// TIA Portal project "Conveyor_Robot_Backup_01_04_2026_V17" (V17)

(* hardware
DEVICE "S7-1200 station_1"  S7-1200 Station
   slot 0: "Rack_0"  S7-1200 Rack  Rack  V1.0
   slot 1: "PLC_1"  CPU 1214C DC/DC/DC  6ES7 214-1AG40-0XB0  V4.4
   slot 2: "DI 8x24VDC/DQ 8xRelay_1"  SM 1223 DI8/DQ8 x relay  6ES7 223-1PH32-0XB0  V2.0
   slot 3: "DI 8x24VDC/DQ 8xRelay_2"  SM 1223 DI8/DQ8 x relay  6ES7 223-1PH32-0XB0  V2.0
DEVICE "HMI_1"  KTP700 Basic PN
   slot 0: "HMI_1"  KTP700 Basic PN  6AV2 123-2GB03-0AX0  16.0.0.0
   slot 1: "HMI_RT_1"  KTP700 Basic PN  6AV2 123-2GB03-0AX0  16.0.0.0
   slot 5: "HMI_1.IE_CP_1"  PROFINET Interface  16.0.0.0
      slot 1: "PROFINET Interface_1"  PROFINET Interface
         slot 1: "Port_1"  Port
*)

// ===== PLC "PLC_1"  CPU 1214C DC/DC/DC =====

VAR_GLOBAL   // PLC tag table "Default tag table"
   "I_PB_Start" AT %I0.0 : Bool;
   "I_PB_Stop" AT %I0.1 : Bool;
   "I_PB_Emergency" AT %I0.2 : Bool;
   "I_PB_Reset" AT %I0.3 : Bool;
   "I_PB_Auto" AT %I0.4 : Bool;
   "I_Sensor_Entry" AT %I0.5 : Bool;
   "I_Sensor_Weigh" AT %I0.6 : Bool;
   "I_Sensor_Decision" AT %I0.7 : Bool;
   "I_Sensor_Reject" AT %I1.0 : Bool;
   "I_Sensor_Exit" AT %I1.1 : Bool;
   "I_Pusher_Extend" AT %I1.2 : Bool;
   "I_Pusher_Released" AT %I1.3 : Bool;
   "I_OL_EntryMotor" AT %I1.4 : Bool;
   "I_OL_WeighMotor" AT %I1.5 : Bool;
   "I_OL_DecideMotor" AT %I2.0 : Bool;
   "I_OL_RejectMotor" AT %I2.1 : Bool;
   "I_OL_ExitMotor" AT %I2.2 : Bool;
   "I_Robot_Detect" AT %I2.3 : Bool;
   "I_Robot_Moving_X" AT %I2.4 : Bool;
   "I_Robot_Moving_Z" AT %I2.5 : Bool;
   "I_Robot_Rotating" AT %I2.6 : Bool;
   "IW_Weight_Loadcell" AT %ID30 : Real;
   "Q_Motor_Entry" AT %Q0.0 : Bool;
   "Q_Motor_Weigh" AT %Q0.1 : Bool;
   "Q_Motor_Decision" AT %Q0.2 : Bool;
   "Q_Motor_reject" AT %Q0.3 : Bool;
   "Q_Motor_Exit" AT %Q0.4 : Bool;
   "Q_Pusher_Extend" AT %Q0.5 : Bool;
   "Q_Pusher_Release" AT %Q0.6 : Bool;
   "Q_Signal_Red" AT %Q2.0 : Bool;
   "Q_Signal_Yellow" AT %Q0.7 : Bool;
   "Q_Signal_Green" AT %Q2.1 : Bool;
   "Q_Buzzer" AT %Q2.2 : Bool;
   "Q_Robot_Extend_X" AT %Q2.3 : Bool;
   "Q_Robot_Down_Z" AT %Q2.4 : Bool;
   "Q_Robot_Grab" AT %Q2.5 : Bool;
   "Q_Robot_Rotate_CW" AT %Q2.6 : Bool;
   "Q_Robot_Rotate_CCW" AT %Q2.7 : Bool;
   "System_Byte" AT %MB1 : Byte;
   "FirstScan" AT %M1.0 : Bool;
   "DiagStatusUpdate" AT %M1.1 : Bool;
   "AlwaysTRUE" AT %M1.2 : Bool;
   "AlwaysFALSE" AT %M1.3 : Bool;
   "Clock_Byte" AT %MB50 : Byte;
   "Clock_10Hz" AT %M50.0 : Bool;
   "Clock_5Hz" AT %M50.1 : Bool;
   "Clock_2.5Hz" AT %M50.2 : Bool;
   "Clock_2Hz" AT %M50.3 : Bool;
   "Clock_1.25Hz" AT %M50.4 : Bool;
   "Clock_1Hz" AT %M50.5 : Bool;
   "Clock_0.625Hz" AT %M50.6 : Bool;
   "Clock_0.5Hz" AT %M50.7 : Bool;
END_VAR

TYPE "UDT_Box_Data"
   STRUCT
      BoxId : Int;
      Weight : Real;
      Status : Bool;
   END_STRUCT;
END_TYPE

TYPE "UDT_Box_Real_Data"
   STRUCT
      Actual_Weight_Value : Real;
      Accept_Limit_Low : Real;
      Accept_Limit_High : Real;
      Current_Box_ID : Int;
   END_STRUCT;
END_TYPE

TYPE "UDT_Alarm"
   STRUCT
      Active : Bool;
      Acknowledge : Bool;
      Cleared : Bool;
      TimeStamp : DTL;
      Duration : Time;
   END_STRUCT;
END_TYPE

TYPE "UDT_OEE_Data"
   STRUCT
      Availability : Real;
      Quality : Real;
      Overall : Real;
      Rating : String;
      Accept_Ratio : Real;
      Reject_Ratio : Real;
   END_STRUCT;
END_TYPE

// folder: 01_Global_DBs

DATA_BLOCK "DB_Batch_Data"   // DB2
{ S7_Optimized_Access := 'TRUE' }
VERSION : 0.1
   VAR
      Batch_ID : Int;
      Batch_Boxes : Int;
      Accept_Boxes : Int;
      Reject_Boxes : Int;
      Accept_Total_Weight : Real;
      Reject_Total_Weight : Real;
      Batch_Running : Bool;
      Low_Limit_Tag : Real;
      High_Limit_Tag : Real;
      Low_Limit_Tag_1 : Real;
      High_Limit_Tag_1 : Real;
      Real_Box_Data : "UDT_Box_Real_Data";
      OEE_Data : "UDT_OEE_Data";
   END_VAR
BEGIN
   Real_Box_Data.Accept_Limit_Low := 3.0;
   Real_Box_Data.Accept_Limit_High := 6.0;
   Real_Box_Data.Current_Box_ID := 0;
END_DATA_BLOCK

DATA_BLOCK "DB_Alarms"   // DB9
{ S7_Optimized_Access := 'TRUE' }
VERSION : 0.1
   VAR
      Motor_Overload : Struct
         OL_EntryMotor : "UDT_Alarm";
         OL_WeighMotor : "UDT_Alarm";
         OL_DecisionMotor : "UDT_Alarm";
         OL_RejectMotor : "UDT_Alarm";
         OL_ExitMotor : "UDT_Alarm";
      END_STRUCT;
      Jam_Alarm : Struct
         Jam_EntryMotor : "UDT_Alarm";
         Jam_WeighMotor : "UDT_Alarm";
         Jam_DecisionMotor : "UDT_Alarm";
         Jam_RejectMotor : "UDT_Alarm";
         Jam_ExitMotor : "UDT_Alarm";
      END_STRUCT;
      Pusher_Alarm : Struct
         Pusher_Stuck_Extended : "UDT_Alarm";
         Pusher_Stuck_Retracted : "UDT_Alarm";
      END_STRUCT;
      HMI_Alarm : Struct
         Jam_Alarm : Word;
         OL_Alarm : Word;
         System_Alarm : Word;
      END_STRUCT;
      HMI_Ack_All : Bool;
   END_VAR
BEGIN
END_DATA_BLOCK

DATA_BLOCK "DB_System_Status"   // DB12
{ S7_Optimized_Access := 'TRUE' }
VERSION : 0.1
   VAR
      System_Running : Bool;
      Enable_Entry : Bool;
      Enable_Weigh : Bool;
      Enable_Decision : Bool;
      Enable_Reject : Bool;
      Enable_Exit : Bool;
      Enable_Robot : Bool;
      Jam_Detected : Struct
         Entry_Jam_Detected : Bool;
         Weigh_Jam_Detected : Bool;
         Decision_Jam_Detected : Bool;
         Reject_Jam_Detected : Bool;
         Exit_Jam_Detected : Bool;
      END_STRUCT;
   END_VAR
BEGIN
END_DATA_BLOCK

// folder: 04_Application_Blocks

DATA_BLOCK "Motor_Control_DB_Entry"   // DB3
{ S7_Optimized_Access := 'TRUE' }
VERSION : 0.1
// stored: InstanceOfName Motor_Control
"Motor_Control"
BEGIN
END_DATA_BLOCK

DATA_BLOCK "Motor_Control_DB_Weigh"   // DB4
{ S7_Optimized_Access := 'TRUE' }
VERSION : 0.1
// stored: InstanceOfName Motor_Control
"Motor_Control"
BEGIN
END_DATA_BLOCK

DATA_BLOCK "Motor_Control_DB_Decision"   // DB5
{ S7_Optimized_Access := 'TRUE' }
VERSION : 0.1
// stored: InstanceOfName Motor_Control
"Motor_Control"
BEGIN
END_DATA_BLOCK

DATA_BLOCK "Motor_Control_DB_Exit"   // DB6
{ S7_Optimized_Access := 'TRUE' }
VERSION : 0.1
// stored: InstanceOfName Motor_Control
"Motor_Control"
BEGIN
END_DATA_BLOCK

DATA_BLOCK "Reject_Conveyor_Control_DB"   // DB7
{ S7_Optimized_Access := 'TRUE' }
VERSION : 0.1
// stored: InstanceOfName Reject_Conveyor_Control
"Reject_Conveyor_Control"
BEGIN
END_DATA_BLOCK

DATA_BLOCK "Arm_Pick_&_Place_DB"   // DB8
{ S7_Optimized_Access := 'TRUE' }
VERSION : 0.1
// stored: InstanceOfName Arm_Pick_&_Place
"Arm_Pick_&_Place"
BEGIN
END_DATA_BLOCK

// folder: 06_IO_Mapping

DATA_BLOCK "DB_IO_Mapping"   // DB1
{ S7_Optimized_Access := 'TRUE' }
VERSION : 0.1
   VAR
      Input : Struct
         I_PB_Start : Bool;
         I_PB_Stop : Bool;
         I_PB_Emergency : Bool;
         I_PB_Reset : Bool;
         I_PB_Auto : Bool;
         I_Sensor_Entry : Bool;
         I_Sensor_Weigh : Bool;
         I_Sensor_Decision : Bool;
         I_Sensor_Reject : Bool;
         I_Sensor_Exit : Bool;
         I_Pusher_Extend : Bool;
         I_Pusher_Released : Bool;
         I_OL_EntryMotor : Bool;
         I_OL_WeighMotor : Bool;
         I_OL_DecideMotor : Bool;
         I_OL_RejectMotor : Bool;
         I_OL_ExitMotor : Bool;
         I_Robot_Detect : Bool;
         I_Robot_Moving_X : Bool;
         I_Robot_Moving_Z : Bool;
         I_Robot_Rotating : Bool;
         IW_Weight_Loadcell : Real;
      END_STRUCT;
      Output : Struct
         Q_Motor_Entry : Bool;
         Q_Motor_Weigh : Bool;
         Q_Motor_Decision : Bool;
         Q_Motor_reject : Bool;
         Q_Motor_Exit : Bool;
         Q_Pusher_Extend : Bool;
         Q_Pusher_Release : Bool;
         Q_Signal_Red : Bool;
         Q_Signal_Yellow : Bool;
         Q_Signal_Green : Bool;
         Q_Buzzer : Bool;
         Q_Robot_Extend_X : Bool;
         Q_Robot_Down_Z : Bool;
         Q_Robot_Grab : Bool;
         Q_Robot_Rotate_CW : Bool;
         Q_Robot_Rotate_CCW : Bool;
      END_STRUCT;
      Parameter : Struct
         M_START : Bool;
      END_STRUCT;
   END_VAR
BEGIN
END_DATA_BLOCK

// folder: System blocks/Program resources

DATA_BLOCK "IEC_Timer_0_DB_1"   // DB10
{ S7_Optimized_Access := 'TRUE' }
AUTHOR : Simatic
FAMILY : IEC
NAME : IEC_TMR
VERSION : 1.0
// stored: InstanceOfName IEC_TIMER
"IEC_TIMER"
BEGIN
END_DATA_BLOCK

// folder: 00_System_Blocks

ORGANIZATION_BLOCK "Main"   // OB1, LAD, ProgramCycle
TITLE = "Main Program Sweep (Cycle)"
{ S7_Optimized_Access := 'TRUE' }
VERSION : 0.1
   VAR_INPUT
      Initial_Call : Bool;   // Initial call of this OB
      Remanence : Bool;   // =True, if remanent data are available
   END_VAR
BEGIN

REGION Network 1: Factory IO Interface
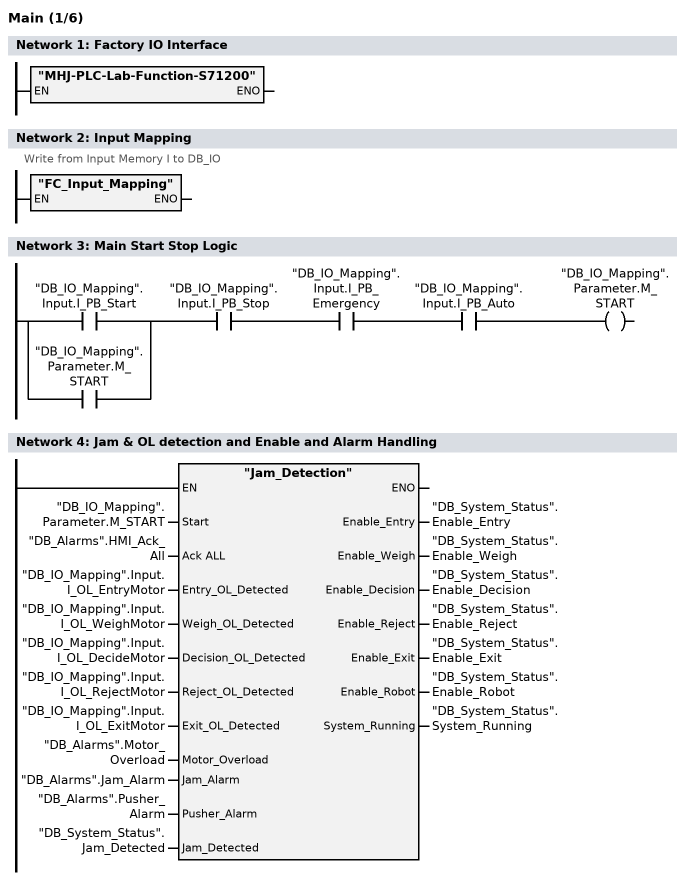
   RUNG wire#powerrail
      "MHJ-PLC-Lab-Function-S71200"()
   END_RUNG
   // the same network as SCL:
   "MHJ-PLC-Lab-Function-S71200"();
END_REGION

REGION Network 2: Input Mapping
   // Write from Input Memory I to DB_IO
   RUNG wire#powerrail
      "FC_Input_Mapping"()
   END_RUNG
   // the same network as SCL:
   "FC_Input_Mapping"();
END_REGION

REGION Network 3: Main Start Stop Logic
   RUNG wire#powerrail
      Contact( "DB_IO_Mapping".Input.I_PB_Start )
      wire#w1
      Contact( "DB_IO_Mapping".Input.I_PB_Stop )
      Contact( "DB_IO_Mapping".Input.I_PB_Emergency )
      Contact( "DB_IO_Mapping".Input.I_PB_Auto )
      Coil( "DB_IO_Mapping".Parameter.M_START )
   END_RUNG
   RUNG wire#powerrail
      Contact( "DB_IO_Mapping".Parameter.M_START )
   END_RUNG wire#w1
   // the same network as SCL:
   "DB_IO_Mapping".Parameter.M_START := ("DB_IO_Mapping".Input.I_PB_Start OR "DB_IO_Mapping".Parameter.M_START) AND "DB_IO_Mapping".Input.I_PB_Stop AND "DB_IO_Mapping".Input.I_PB_Emergency AND "DB_IO_Mapping".Input.I_PB_Auto;
END_REGION

REGION Network 4: Jam & OL detection and Enable and Alarm Handling
   RUNG wire#powerrail
      "Jam_Detection"(Start := "DB_IO_Mapping".Parameter.M_START, "Ack ALL" := "DB_Alarms".HMI_Ack_All, Entry_OL_Detected := "DB_IO_Mapping".Input.I_OL_EntryMotor, Weigh_OL_Detected := "DB_IO_Mapping".Input.I_OL_WeighMotor, Decision_OL_Detected := "DB_IO_Mapping".Input.I_OL_DecideMotor, Reject_OL_Detected := "DB_IO_Mapping".Input.I_OL_RejectMotor, Exit_OL_Detected := "DB_IO_Mapping".Input.I_OL_ExitMotor, Motor_Overload := "DB_Alarms".Motor_Overload, Jam_Alarm := "DB_Alarms".Jam_Alarm, Pusher_Alarm := "DB_Alarms".Pusher_Alarm, Jam_Detected := "DB_System_Status".Jam_Detected, Enable_Entry => "DB_System_Status".Enable_Entry, Enable_Weigh => "DB_System_Status".Enable_Weigh, Enable_Decision => "DB_System_Status".Enable_Decision, Enable_Reject => "DB_System_Status".Enable_Reject, Enable_Exit => "DB_System_Status".Enable_Exit, Enable_Robot => "DB_System_Status".Enable_Robot, System_Running => "DB_System_Status".System_Running)
   END_RUNG
   // the same network as SCL:
   "Jam_Detection"(Start := "DB_IO_Mapping".Parameter.M_START,
                   "Ack ALL" := "DB_Alarms".HMI_Ack_All,
                   Entry_OL_Detected := "DB_IO_Mapping".Input.I_OL_EntryMotor,
                   Weigh_OL_Detected := "DB_IO_Mapping".Input.I_OL_WeighMotor,
                   Decision_OL_Detected := "DB_IO_Mapping".Input.I_OL_DecideMotor,
                   Reject_OL_Detected := "DB_IO_Mapping".Input.I_OL_RejectMotor,
                   Exit_OL_Detected := "DB_IO_Mapping".Input.I_OL_ExitMotor,
                   Motor_Overload := "DB_Alarms".Motor_Overload,
                   Jam_Alarm := "DB_Alarms".Jam_Alarm,
                   Pusher_Alarm := "DB_Alarms".Pusher_Alarm,
                   Jam_Detected := "DB_System_Status".Jam_Detected,
                   Enable_Entry => "DB_System_Status".Enable_Entry,
                   Enable_Weigh => "DB_System_Status".Enable_Weigh,
                   Enable_Decision => "DB_System_Status".Enable_Decision,
                   Enable_Reject => "DB_System_Status".Enable_Reject,
                   Enable_Exit => "DB_System_Status".Enable_Exit,
                   Enable_Robot => "DB_System_Status".Enable_Robot,
                   System_Running => "DB_System_Status".System_Running);
END_REGION

REGION Network 5: Entry Conveyor
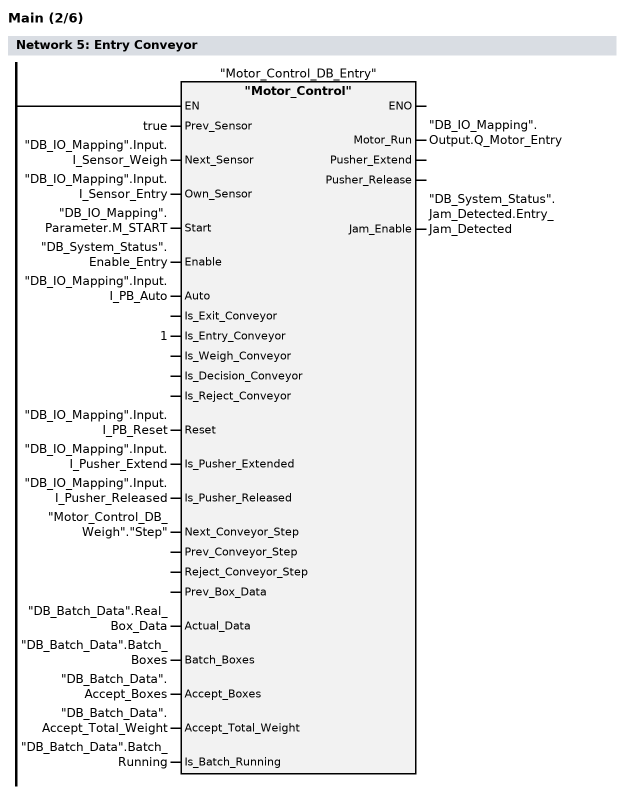
   RUNG wire#powerrail
      "Motor_Control_DB_Entry"(Prev_Sensor := true, Next_Sensor := "DB_IO_Mapping".Input.I_Sensor_Weigh, Own_Sensor := "DB_IO_Mapping".Input.I_Sensor_Entry, Start := "DB_IO_Mapping".Parameter.M_START, Enable := "DB_System_Status".Enable_Entry, Auto := "DB_IO_Mapping".Input.I_PB_Auto, Is_Exit_Conveyor :=, Is_Entry_Conveyor := 1, Is_Weigh_Conveyor :=, Is_Decision_Conveyor :=, Is_Reject_Conveyor :=, Reset := "DB_IO_Mapping".Input.I_PB_Reset, Is_Pusher_Extended := "DB_IO_Mapping".Input.I_Pusher_Extend, Is_Pusher_Released := "DB_IO_Mapping".Input.I_Pusher_Released, Next_Conveyor_Step := "Motor_Control_DB_Weigh"."Step", Prev_Conveyor_Step :=, Reject_Conveyor_Step :=, Prev_Box_Data :=, Actual_Data := "DB_Batch_Data".Real_Box_Data, Batch_Boxes := "DB_Batch_Data".Batch_Boxes, Accept_Boxes := "DB_Batch_Data".Accept_Boxes, Accept_Total_Weight := "DB_Batch_Data".Accept_Total_Weight, Is_Batch_Running := "DB_Batch_Data".Batch_Running, Motor_Run => "DB_IO_Mapping".Output.Q_Motor_Entry, Pusher_Extend =>, Pusher_Release =>, Jam_Enable => "DB_System_Status".Jam_Detected.Entry_Jam_Detected)
   END_RUNG
   // the same network as SCL:
   "Motor_Control_DB_Entry"(Prev_Sensor := true,   // "Motor_Control"
                           Next_Sensor := "DB_IO_Mapping".Input.I_Sensor_Weigh,
                           Own_Sensor := "DB_IO_Mapping".Input.I_Sensor_Entry,
                           Start := "DB_IO_Mapping".Parameter.M_START,
                           Enable := "DB_System_Status".Enable_Entry,
                           Auto := "DB_IO_Mapping".Input.I_PB_Auto,
                           Is_Entry_Conveyor := 1,
                           Reset := "DB_IO_Mapping".Input.I_PB_Reset,
                           Is_Pusher_Extended := "DB_IO_Mapping".Input.I_Pusher_Extend,
                           Is_Pusher_Released := "DB_IO_Mapping".Input.I_Pusher_Released,
                           Next_Conveyor_Step := "Motor_Control_DB_Weigh"."Step",
                           Actual_Data := "DB_Batch_Data".Real_Box_Data,
                           Batch_Boxes := "DB_Batch_Data".Batch_Boxes,
                           Accept_Boxes := "DB_Batch_Data".Accept_Boxes,
                           Accept_Total_Weight := "DB_Batch_Data".Accept_Total_Weight,
                           Is_Batch_Running := "DB_Batch_Data".Batch_Running,
                           Motor_Run => "DB_IO_Mapping".Output.Q_Motor_Entry,
                           Jam_Enable => "DB_System_Status".Jam_Detected.Entry_Jam_Detected);
END_REGION

REGION Network 6: Weigh Conveyor
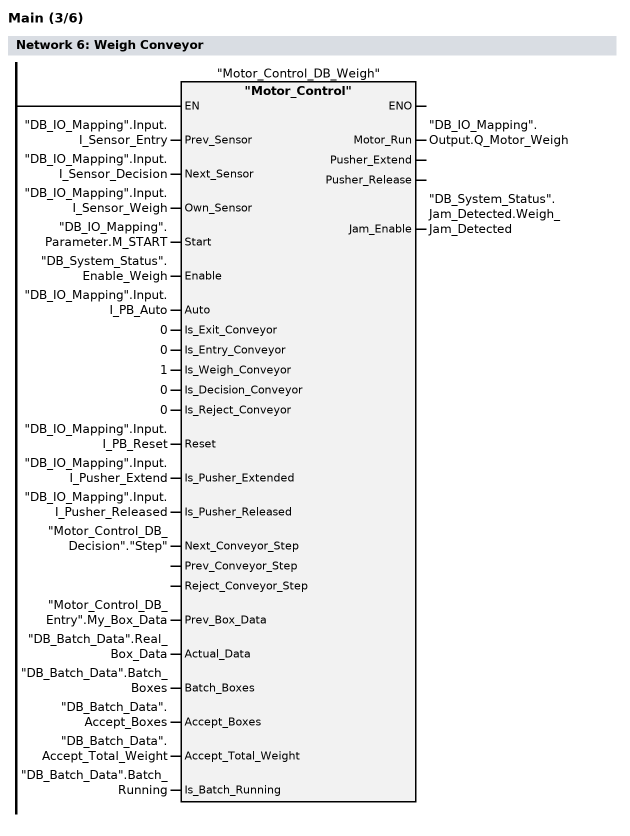
   RUNG wire#powerrail
      "Motor_Control_DB_Weigh"(Prev_Sensor := "DB_IO_Mapping".Input.I_Sensor_Entry, Next_Sensor := "DB_IO_Mapping".Input.I_Sensor_Decision, Own_Sensor := "DB_IO_Mapping".Input.I_Sensor_Weigh, Start := "DB_IO_Mapping".Parameter.M_START, Enable := "DB_System_Status".Enable_Weigh, Auto := "DB_IO_Mapping".Input.I_PB_Auto, Is_Exit_Conveyor := 0, Is_Entry_Conveyor := 0, Is_Weigh_Conveyor := 1, Is_Decision_Conveyor := 0, Is_Reject_Conveyor := 0, Reset := "DB_IO_Mapping".Input.I_PB_Reset, Is_Pusher_Extended := "DB_IO_Mapping".Input.I_Pusher_Extend, Is_Pusher_Released := "DB_IO_Mapping".Input.I_Pusher_Released, Next_Conveyor_Step := "Motor_Control_DB_Decision"."Step", Prev_Conveyor_Step :=, Reject_Conveyor_Step :=, Prev_Box_Data := "Motor_Control_DB_Entry".My_Box_Data, Actual_Data := "DB_Batch_Data".Real_Box_Data, Batch_Boxes := "DB_Batch_Data".Batch_Boxes, Accept_Boxes := "DB_Batch_Data".Accept_Boxes, Accept_Total_Weight := "DB_Batch_Data".Accept_Total_Weight, Is_Batch_Running := "DB_Batch_Data".Batch_Running, Motor_Run => "DB_IO_Mapping".Output.Q_Motor_Weigh, Pusher_Extend =>, Pusher_Release =>, Jam_Enable => "DB_System_Status".Jam_Detected.Weigh_Jam_Detected)
   END_RUNG
   // the same network as SCL:
   "Motor_Control_DB_Weigh"(Prev_Sensor := "DB_IO_Mapping".Input.I_Sensor_Entry,   // "Motor_Control"
                           Next_Sensor := "DB_IO_Mapping".Input.I_Sensor_Decision,
                           Own_Sensor := "DB_IO_Mapping".Input.I_Sensor_Weigh,
                           Start := "DB_IO_Mapping".Parameter.M_START,
                           Enable := "DB_System_Status".Enable_Weigh,
                           Auto := "DB_IO_Mapping".Input.I_PB_Auto,
                           Is_Exit_Conveyor := 0,
                           Is_Entry_Conveyor := 0,
                           Is_Weigh_Conveyor := 1,
                           Is_Decision_Conveyor := 0,
                           Is_Reject_Conveyor := 0,
                           Reset := "DB_IO_Mapping".Input.I_PB_Reset,
                           Is_Pusher_Extended := "DB_IO_Mapping".Input.I_Pusher_Extend,
                           Is_Pusher_Released := "DB_IO_Mapping".Input.I_Pusher_Released,
                           Next_Conveyor_Step := "Motor_Control_DB_Decision"."Step",
                           Prev_Box_Data := "Motor_Control_DB_Entry".My_Box_Data,
                           Actual_Data := "DB_Batch_Data".Real_Box_Data,
                           Batch_Boxes := "DB_Batch_Data".Batch_Boxes,
                           Accept_Boxes := "DB_Batch_Data".Accept_Boxes,
                           Accept_Total_Weight := "DB_Batch_Data".Accept_Total_Weight,
                           Is_Batch_Running := "DB_Batch_Data".Batch_Running,
                           Motor_Run => "DB_IO_Mapping".Output.Q_Motor_Weigh,
                           Jam_Enable => "DB_System_Status".Jam_Detected.Weigh_Jam_Detected);
END_REGION

REGION Network 7: Decision Conveyor
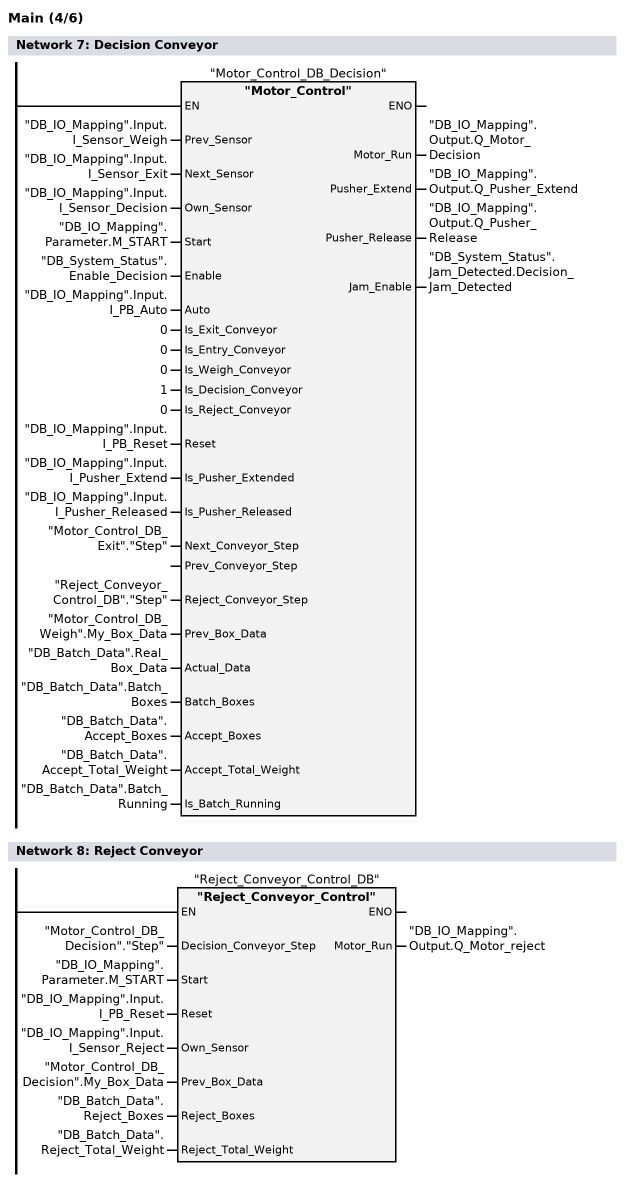
   RUNG wire#powerrail
      "Motor_Control_DB_Decision"(Prev_Sensor := "DB_IO_Mapping".Input.I_Sensor_Weigh, Next_Sensor := "DB_IO_Mapping".Input.I_Sensor_Exit, Own_Sensor := "DB_IO_Mapping".Input.I_Sensor_Decision, Start := "DB_IO_Mapping".Parameter.M_START, Enable := "DB_System_Status".Enable_Decision, Auto := "DB_IO_Mapping".Input.I_PB_Auto, Is_Exit_Conveyor := 0, Is_Entry_Conveyor := 0, Is_Weigh_Conveyor := 0, Is_Decision_Conveyor := 1, Is_Reject_Conveyor := 0, Reset := "DB_IO_Mapping".Input.I_PB_Reset, Is_Pusher_Extended := "DB_IO_Mapping".Input.I_Pusher_Extend, Is_Pusher_Released := "DB_IO_Mapping".Input.I_Pusher_Released, Next_Conveyor_Step := "Motor_Control_DB_Exit"."Step", Prev_Conveyor_Step :=, Reject_Conveyor_Step := "Reject_Conveyor_Control_DB"."Step", Prev_Box_Data := "Motor_Control_DB_Weigh".My_Box_Data, Actual_Data := "DB_Batch_Data".Real_Box_Data, Batch_Boxes := "DB_Batch_Data".Batch_Boxes, Accept_Boxes := "DB_Batch_Data".Accept_Boxes, Accept_Total_Weight := "DB_Batch_Data".Accept_Total_Weight, Is_Batch_Running := "DB_Batch_Data".Batch_Running, Motor_Run => "DB_IO_Mapping".Output.Q_Motor_Decision, Pusher_Extend => "DB_IO_Mapping".Output.Q_Pusher_Extend, Pusher_Release => "DB_IO_Mapping".Output.Q_Pusher_Release, Jam_Enable => "DB_System_Status".Jam_Detected.Decision_Jam_Detected)
   END_RUNG
   // the same network as SCL:
   "Motor_Control_DB_Decision"(Prev_Sensor := "DB_IO_Mapping".Input.I_Sensor_Weigh,   // "Motor_Control"
                           Next_Sensor := "DB_IO_Mapping".Input.I_Sensor_Exit,
                           Own_Sensor := "DB_IO_Mapping".Input.I_Sensor_Decision,
                           Start := "DB_IO_Mapping".Parameter.M_START,
                           Enable := "DB_System_Status".Enable_Decision,
                           Auto := "DB_IO_Mapping".Input.I_PB_Auto,
                           Is_Exit_Conveyor := 0,
                           Is_Entry_Conveyor := 0,
                           Is_Weigh_Conveyor := 0,
                           Is_Decision_Conveyor := 1,
                           Is_Reject_Conveyor := 0,
                           Reset := "DB_IO_Mapping".Input.I_PB_Reset,
                           Is_Pusher_Extended := "DB_IO_Mapping".Input.I_Pusher_Extend,
                           Is_Pusher_Released := "DB_IO_Mapping".Input.I_Pusher_Released,
                           Next_Conveyor_Step := "Motor_Control_DB_Exit"."Step",
                           Reject_Conveyor_Step := "Reject_Conveyor_Control_DB"."Step",
                           Prev_Box_Data := "Motor_Control_DB_Weigh".My_Box_Data,
                           Actual_Data := "DB_Batch_Data".Real_Box_Data,
                           Batch_Boxes := "DB_Batch_Data".Batch_Boxes,
                           Accept_Boxes := "DB_Batch_Data".Accept_Boxes,
                           Accept_Total_Weight := "DB_Batch_Data".Accept_Total_Weight,
                           Is_Batch_Running := "DB_Batch_Data".Batch_Running,
                           Motor_Run => "DB_IO_Mapping".Output.Q_Motor_Decision,
                           Pusher_Extend => "DB_IO_Mapping".Output.Q_Pusher_Extend,
                           Pusher_Release => "DB_IO_Mapping".Output.Q_Pusher_Release,
                           Jam_Enable => "DB_System_Status".Jam_Detected.Decision_Jam_Detected);
END_REGION

REGION Network 8: Reject Conveyor
   RUNG wire#powerrail
      "Reject_Conveyor_Control_DB"(Decision_Conveyor_Step := "Motor_Control_DB_Decision"."Step", Start := "DB_IO_Mapping".Parameter.M_START, Reset := "DB_IO_Mapping".Input.I_PB_Reset, Own_Sensor := "DB_IO_Mapping".Input.I_Sensor_Reject, Prev_Box_Data := "Motor_Control_DB_Decision".My_Box_Data, Reject_Boxes := "DB_Batch_Data".Reject_Boxes, Reject_Total_Weight := "DB_Batch_Data".Reject_Total_Weight, Motor_Run => "DB_IO_Mapping".Output.Q_Motor_reject)
   END_RUNG
   // the same network as SCL:
   "Reject_Conveyor_Control_DB"(Decision_Conveyor_Step := "Motor_Control_DB_Decision"."Step",   // "Reject_Conveyor_Control"
                           Start := "DB_IO_Mapping".Parameter.M_START,
                           Reset := "DB_IO_Mapping".Input.I_PB_Reset,
                           Own_Sensor := "DB_IO_Mapping".Input.I_Sensor_Reject,
                           Prev_Box_Data := "Motor_Control_DB_Decision".My_Box_Data,
                           Reject_Boxes := "DB_Batch_Data".Reject_Boxes,
                           Reject_Total_Weight := "DB_Batch_Data".Reject_Total_Weight,
                           Motor_Run => "DB_IO_Mapping".Output.Q_Motor_reject);
END_REGION

REGION Network 9: Exit Conveyor
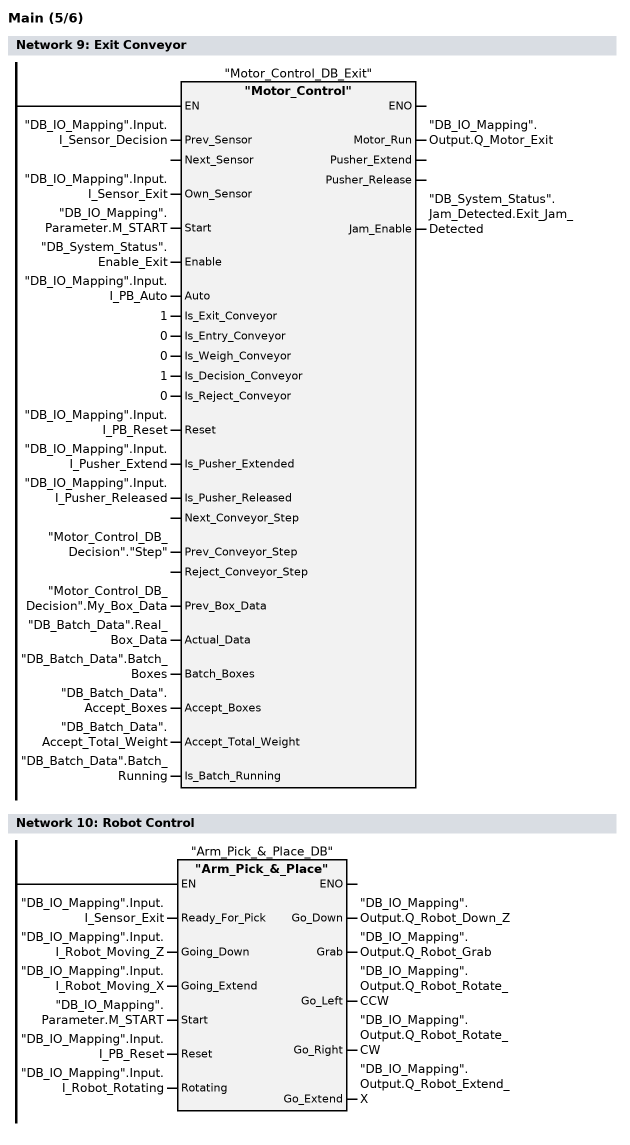
   RUNG wire#powerrail
      "Motor_Control_DB_Exit"(Prev_Sensor := "DB_IO_Mapping".Input.I_Sensor_Decision, Next_Sensor :=, Own_Sensor := "DB_IO_Mapping".Input.I_Sensor_Exit, Start := "DB_IO_Mapping".Parameter.M_START, Enable := "DB_System_Status".Enable_Exit, Auto := "DB_IO_Mapping".Input.I_PB_Auto, Is_Exit_Conveyor := 1, Is_Entry_Conveyor := 0, Is_Weigh_Conveyor := 0, Is_Decision_Conveyor := 1, Is_Reject_Conveyor := 0, Reset := "DB_IO_Mapping".Input.I_PB_Reset, Is_Pusher_Extended := "DB_IO_Mapping".Input.I_Pusher_Extend, Is_Pusher_Released := "DB_IO_Mapping".Input.I_Pusher_Released, Next_Conveyor_Step :=, Prev_Conveyor_Step := "Motor_Control_DB_Decision"."Step", Reject_Conveyor_Step :=, Prev_Box_Data := "Motor_Control_DB_Decision".My_Box_Data, Actual_Data := "DB_Batch_Data".Real_Box_Data, Batch_Boxes := "DB_Batch_Data".Batch_Boxes, Accept_Boxes := "DB_Batch_Data".Accept_Boxes, Accept_Total_Weight := "DB_Batch_Data".Accept_Total_Weight, Is_Batch_Running := "DB_Batch_Data".Batch_Running, Motor_Run => "DB_IO_Mapping".Output.Q_Motor_Exit, Pusher_Extend =>, Pusher_Release =>, Jam_Enable => "DB_System_Status".Jam_Detected.Exit_Jam_Detected)
   END_RUNG
   // the same network as SCL:
   "Motor_Control_DB_Exit"(Prev_Sensor := "DB_IO_Mapping".Input.I_Sensor_Decision,   // "Motor_Control"
                           Own_Sensor := "DB_IO_Mapping".Input.I_Sensor_Exit,
                           Start := "DB_IO_Mapping".Parameter.M_START,
                           Enable := "DB_System_Status".Enable_Exit,
                           Auto := "DB_IO_Mapping".Input.I_PB_Auto,
                           Is_Exit_Conveyor := 1,
                           Is_Entry_Conveyor := 0,
                           Is_Weigh_Conveyor := 0,
                           Is_Decision_Conveyor := 1,
                           Is_Reject_Conveyor := 0,
                           Reset := "DB_IO_Mapping".Input.I_PB_Reset,
                           Is_Pusher_Extended := "DB_IO_Mapping".Input.I_Pusher_Extend,
                           Is_Pusher_Released := "DB_IO_Mapping".Input.I_Pusher_Released,
                           Prev_Conveyor_Step := "Motor_Control_DB_Decision"."Step",
                           Prev_Box_Data := "Motor_Control_DB_Decision".My_Box_Data,
                           Actual_Data := "DB_Batch_Data".Real_Box_Data,
                           Batch_Boxes := "DB_Batch_Data".Batch_Boxes,
                           Accept_Boxes := "DB_Batch_Data".Accept_Boxes,
                           Accept_Total_Weight := "DB_Batch_Data".Accept_Total_Weight,
                           Is_Batch_Running := "DB_Batch_Data".Batch_Running,
                           Motor_Run => "DB_IO_Mapping".Output.Q_Motor_Exit,
                           Jam_Enable => "DB_System_Status".Jam_Detected.Exit_Jam_Detected);
END_REGION

REGION Network 10: Robot Control
   RUNG wire#powerrail
      "Arm_Pick_&_Place_DB"(Ready_For_Pick := "DB_IO_Mapping".Input.I_Sensor_Exit, Going_Down := "DB_IO_Mapping".Input.I_Robot_Moving_Z, Going_Extend := "DB_IO_Mapping".Input.I_Robot_Moving_X, Start := "DB_IO_Mapping".Parameter.M_START, Reset := "DB_IO_Mapping".Input.I_PB_Reset, Rotating := "DB_IO_Mapping".Input.I_Robot_Rotating, Go_Down => "DB_IO_Mapping".Output.Q_Robot_Down_Z, Grab => "DB_IO_Mapping".Output.Q_Robot_Grab, Go_Left => "DB_IO_Mapping".Output.Q_Robot_Rotate_CCW, Go_Right => "DB_IO_Mapping".Output.Q_Robot_Rotate_CW, Go_Extend => "DB_IO_Mapping".Output.Q_Robot_Extend_X)
   END_RUNG
   // the same network as SCL:
   "Arm_Pick_&_Place_DB"(Ready_For_Pick := "DB_IO_Mapping".Input.I_Sensor_Exit,   // "Arm_Pick_&_Place"
                         Going_Down := "DB_IO_Mapping".Input.I_Robot_Moving_Z,
                         Going_Extend := "DB_IO_Mapping".Input.I_Robot_Moving_X,
                         Start := "DB_IO_Mapping".Parameter.M_START,
                         Reset := "DB_IO_Mapping".Input.I_PB_Reset,
                         Rotating := "DB_IO_Mapping".Input.I_Robot_Rotating,
                         Go_Down => "DB_IO_Mapping".Output.Q_Robot_Down_Z,
                         Grab => "DB_IO_Mapping".Output.Q_Robot_Grab,
                         Go_Left => "DB_IO_Mapping".Output.Q_Robot_Rotate_CCW,
                         Go_Right => "DB_IO_Mapping".Output.Q_Robot_Rotate_CW,
                         Go_Extend => "DB_IO_Mapping".Output.Q_Robot_Extend_X);
END_REGION

REGION Network 11: HMI Interface Fc
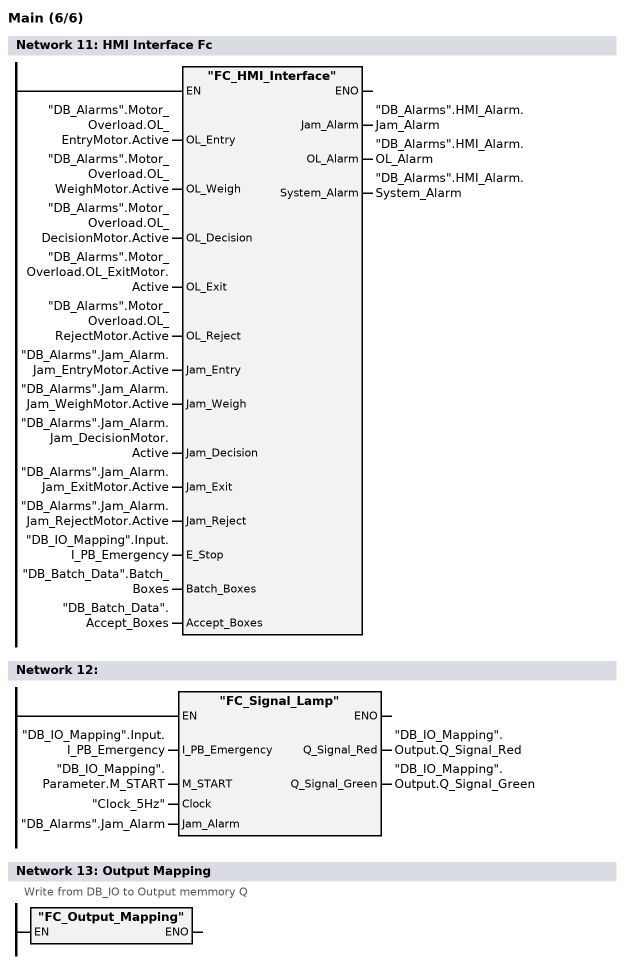
   RUNG wire#powerrail
      "FC_HMI_Interface"(OL_Entry := "DB_Alarms".Motor_Overload.OL_EntryMotor.Active, OL_Weigh := "DB_Alarms".Motor_Overload.OL_WeighMotor.Active, OL_Decision := "DB_Alarms".Motor_Overload.OL_DecisionMotor.Active, OL_Exit := "DB_Alarms".Motor_Overload.OL_ExitMotor.Active, OL_Reject := "DB_Alarms".Motor_Overload.OL_RejectMotor.Active, Jam_Entry := "DB_Alarms".Jam_Alarm.Jam_EntryMotor.Active, Jam_Weigh := "DB_Alarms".Jam_Alarm.Jam_WeighMotor.Active, Jam_Decision := "DB_Alarms".Jam_Alarm.Jam_DecisionMotor.Active, Jam_Exit := "DB_Alarms".Jam_Alarm.Jam_ExitMotor.Active, Jam_Reject := "DB_Alarms".Jam_Alarm.Jam_RejectMotor.Active, E_Stop := "DB_IO_Mapping".Input.I_PB_Emergency, Batch_Boxes := "DB_Batch_Data".Batch_Boxes, Accept_Boxes := "DB_Batch_Data".Accept_Boxes, Jam_Alarm => "DB_Alarms".HMI_Alarm.Jam_Alarm, OL_Alarm => "DB_Alarms".HMI_Alarm.OL_Alarm, System_Alarm => "DB_Alarms".HMI_Alarm.System_Alarm)
   END_RUNG
   // the same network as SCL:
   "FC_HMI_Interface"(OL_Entry := "DB_Alarms".Motor_Overload.OL_EntryMotor.Active,
                      OL_Weigh := "DB_Alarms".Motor_Overload.OL_WeighMotor.Active,
                      OL_Decision := "DB_Alarms".Motor_Overload.OL_DecisionMotor.Active,
                      OL_Exit := "DB_Alarms".Motor_Overload.OL_ExitMotor.Active,
                      OL_Reject := "DB_Alarms".Motor_Overload.OL_RejectMotor.Active,
                      Jam_Entry := "DB_Alarms".Jam_Alarm.Jam_EntryMotor.Active,
                      Jam_Weigh := "DB_Alarms".Jam_Alarm.Jam_WeighMotor.Active,
                      Jam_Decision := "DB_Alarms".Jam_Alarm.Jam_DecisionMotor.Active,
                      Jam_Exit := "DB_Alarms".Jam_Alarm.Jam_ExitMotor.Active,
                      Jam_Reject := "DB_Alarms".Jam_Alarm.Jam_RejectMotor.Active,
                      E_Stop := "DB_IO_Mapping".Input.I_PB_Emergency,
                      Batch_Boxes := "DB_Batch_Data".Batch_Boxes,
                      Accept_Boxes := "DB_Batch_Data".Accept_Boxes,
                      Jam_Alarm => "DB_Alarms".HMI_Alarm.Jam_Alarm,
                      OL_Alarm => "DB_Alarms".HMI_Alarm.OL_Alarm,
                      System_Alarm => "DB_Alarms".HMI_Alarm.System_Alarm);
END_REGION

REGION Network 12
   RUNG wire#powerrail
      "FC_Signal_Lamp"(I_PB_Emergency := "DB_IO_Mapping".Input.I_PB_Emergency, M_START := "DB_IO_Mapping".Parameter.M_START, Clock := "Clock_5Hz", Jam_Alarm := "DB_Alarms".Jam_Alarm, Q_Signal_Red => "DB_IO_Mapping".Output.Q_Signal_Red, Q_Signal_Green => "DB_IO_Mapping".Output.Q_Signal_Green)
   END_RUNG
   // the same network as SCL:
   "FC_Signal_Lamp"(I_PB_Emergency := "DB_IO_Mapping".Input.I_PB_Emergency,
                    M_START := "DB_IO_Mapping".Parameter.M_START,
                    Clock := "Clock_5Hz",
                    Jam_Alarm := "DB_Alarms".Jam_Alarm,
                    Q_Signal_Red => "DB_IO_Mapping".Output.Q_Signal_Red,
                    Q_Signal_Green => "DB_IO_Mapping".Output.Q_Signal_Green);
END_REGION

REGION Network 13: Output Mapping
   // Write from DB_IO to Output memmory Q
   RUNG wire#powerrail
      "FC_Output_Mapping"()
   END_RUNG
   // the same network as SCL:
   "FC_Output_Mapping"();
END_REGION
END_ORGANIZATION_BLOCK

ORGANIZATION_BLOCK "Time error interrupt"   // OB80, SCL, TimeErrorInterrupt
{ S7_Optimized_Access := 'TRUE' }
VERSION : 0.1
   VAR_INPUT
      Fault_ID : Byte;   // Fault identifier
      Csg_OBnr : OB_Any;   // Number of OB causing the error
      Csg_Prio : UInt;   // Priority of OB causing the error
   END_VAR
BEGIN

   "FC_Clear_O/P"(Output := "DB_IO_Mapping".Output);

   "DB_Alarms".HMI_Alarm.System_Alarm.%X2 := TRUE;//Set ALarm of System ALram bit 1 for HMI indication

   "DB_System_Status".System_Running := FALSE; //System run stop
END_ORGANIZATION_BLOCK

ORGANIZATION_BLOCK "Startup"   // OB100, LAD, Startup
TITLE = "Complete Restart"
{ S7_Optimized_Access := 'TRUE' }
VERSION : 0.1
   VAR_INPUT
      LostRetentive : Bool;   // True if retentive data are lost
      LostRTC : Bool;   // True if date and time are lost
   END_VAR
BEGIN

REGION Network 1: Initial Value Load
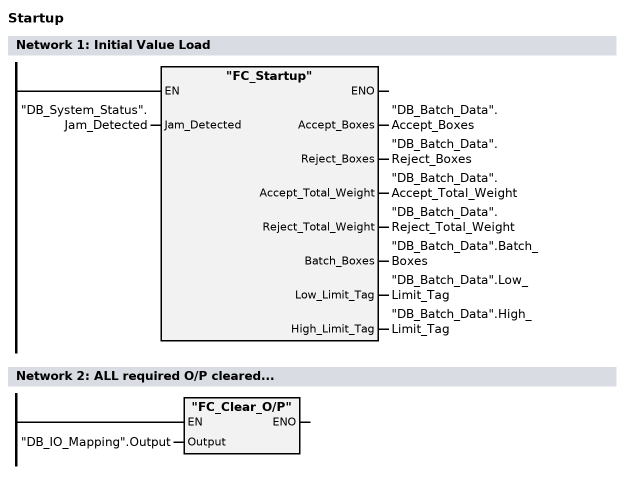
   RUNG wire#powerrail
      "FC_Startup"(Jam_Detected := "DB_System_Status".Jam_Detected, Accept_Boxes => "DB_Batch_Data".Accept_Boxes, Reject_Boxes => "DB_Batch_Data".Reject_Boxes, Accept_Total_Weight => "DB_Batch_Data".Accept_Total_Weight, Reject_Total_Weight => "DB_Batch_Data".Reject_Total_Weight, Batch_Boxes => "DB_Batch_Data".Batch_Boxes, Low_Limit_Tag => "DB_Batch_Data".Low_Limit_Tag, High_Limit_Tag => "DB_Batch_Data".High_Limit_Tag)
   END_RUNG
   // the same network as SCL:
   "FC_Startup"(Jam_Detected := "DB_System_Status".Jam_Detected,
                Accept_Boxes => "DB_Batch_Data".Accept_Boxes,
                Reject_Boxes => "DB_Batch_Data".Reject_Boxes,
                Accept_Total_Weight => "DB_Batch_Data".Accept_Total_Weight,
                Reject_Total_Weight => "DB_Batch_Data".Reject_Total_Weight,
                Batch_Boxes => "DB_Batch_Data".Batch_Boxes,
                Low_Limit_Tag => "DB_Batch_Data".Low_Limit_Tag,
                High_Limit_Tag => "DB_Batch_Data".High_Limit_Tag);
END_REGION

REGION Network 2: ALL required O/P cleared...
   RUNG wire#powerrail
      "FC_Clear_O/P"(Output := "DB_IO_Mapping".Output)
   END_RUNG
   // the same network as SCL:
   "FC_Clear_O/P"(Output := "DB_IO_Mapping".Output);
END_REGION
END_ORGANIZATION_BLOCK

// folder: 02_Library_FBs

FUNCTION_BLOCK "Motor_Control"   // FB1, SCL
{ S7_Optimized_Access := 'TRUE' }
VERSION : 0.1
   VAR_INPUT
      Prev_Sensor : Bool;
      Next_Sensor : Bool;
      Own_Sensor : Bool;
      Start : Bool;
      Enable : Bool;
      Auto : Bool;
      Is_Exit_Conveyor : Bool;
      Is_Entry_Conveyor : Bool;
      Is_Weigh_Conveyor : Bool;
      Is_Decision_Conveyor : Bool;
      Is_Reject_Conveyor : Bool;
      Reset : Bool;
      Is_Pusher_Extended : Bool;
      Is_Pusher_Released : Bool;
      Next_Conveyor_Step : Int;
      Prev_Conveyor_Step : Int;
      Reject_Conveyor_Step : Int;
      Prev_Box_Data : "UDT_Box_Data";
      Actual_Data : "UDT_Box_Real_Data";
   END_VAR
   VAR_OUTPUT
      Motor_Run : Bool;
      Pusher_Extend : Bool;
      Pusher_Release : Bool;
      Jam_Enable : Bool;
   END_VAR
   VAR_IN_OUT
      Batch_Boxes : Int;
      Accept_Boxes : Int;
      Accept_Total_Weight : Real;
      Is_Batch_Running : Bool;
   END_VAR
   VAR
      "Step" : Int;
      Timer_Done : Bool;
      Timer_Enabale : Bool;
      Timer_ET : Time;
      Timer_Started : Bool;
      Timer_OFF_Dealy_Enable : Bool;
      My_Box_Data : "UDT_Box_Data";
      Jam_Detection_Timer : TON_TIME;
   END_VAR
BEGIN
   IF #Batch_Boxes > #Accept_Boxes THEN
       #Is_Batch_Running := TRUE;
   ELSE
       #Is_Batch_Running := FALSE;
   END_IF;

   IF #Start & #Enable & #Is_Batch_Running THEN

       IF #Is_Weigh_Conveyor THEN
           // Trigger timer only first time in Step 20
           "IEC_Timer_0_DB_1".TON(IN := (#Step = 20),
                                  PT := T#1s,
                                  Q => #Timer_Done,
                                  ET => #Timer_ET);
       END_IF;





       CASE #Step OF
           0: //Sensor at Previous sensor and own sensor is empty...
               #Motor_Run := FALSE;


                   IF #Prev_Sensor & NOT #Own_Sensor THEN
                       #Motor_Run := TRUE;
                       #Step := 10;
                   END_IF;


               ;


           10: // Motor is running till Box reached to it's own sensor
               #Motor_Run := TRUE;

               // Jam detection Logic
               // 
               IF #Is_Exit_Conveyor THEN
                   IF #Prev_Conveyor_Step >= 40 THEN
                       #Jam_Detection_Timer(IN := TRUE,
                                            PT := T#6s);
                   END_IF;
               ELSE
                   #Jam_Detection_Timer(IN := TRUE,
                                        PT := T#6s);
               END_IF;

               // #Jam_Detection_Timer(IN := TRUE,
               //                      PT := T#20s);

               IF #Jam_Detection_Timer.Q THEN
                   #Jam_Enable := TRUE;

               END_IF;

               IF #Own_Sensor THEN

                   #Jam_Detection_Timer(IN := FALSE,
                                        PT := T#6s);
                   #Jam_Enable := FALSE;

                   #Motor_Run := FALSE;
                   #Step := 20;
               END_IF;
               ;





           20://As reached to own sensor now motor stop, As here conveyor wise few task needed to perform
               #Motor_Run := FALSE;



               //If Weigh conveyor Than Data of box generation done here
               IF #Is_Weigh_Conveyor & #Timer_Done THEN //First time data feed
                   "FC_WeighScale_Data_Transfer"(Actual_Data := #Actual_Data,
                                                 My_Box_Data => #My_Box_Data);
                   #Step := 30;

                   ;

                   //And If not weigh than previous conveyor data transfer to Own data
               ELSIF NOT #Is_Weigh_Conveyor & NOT #Is_Entry_Conveyor THEN
                   "FC_BoxData_Transfer"(Prev_Box_Data := #Prev_Box_Data,
                                         My_Box_Data => #My_Box_Data);
                   #Step := 30;
                   ;

                   //If Entry conveyor than no data needed so Direct 30
               ELSIF #Is_Entry_Conveyor THEN
                   #Step := 30;
                   ;

                   ;
               END_IF;
               ;


           30: //As Now data transfered so now move to next 
               #Motor_Run := FALSE;


               //If exit conveyor than Robot pick a box, SO Rise accept box and weight and step =0
               IF #Is_Exit_Conveyor THEN
                   IF NOT #Own_Sensor THEN
                       #Accept_Boxes := #Accept_Boxes + 1;
                       #Accept_Total_Weight := #Accept_Total_Weight + #My_Box_Data.Weight;

                       #Step := 0;
                   END_IF;
                   ;
                   ;

                   //If decision conveyor than check accept or reject
               ELSIF #Is_Decision_Conveyor & NOT #My_Box_Data.Status THEN
                   // As decision & status is false so now Pusher Extend here and return back ok...
                   #Pusher_Extend := TRUE;// add off delay time here...
                   #Step := 31;



                   ;

                   //If next conveyor is empty and ready to pick a box than start a motor
               ELSE
                   IF #Own_Sensor & NOT #Next_Sensor & #Next_Conveyor_Step = 10 THEN
                       #Motor_Run := TRUE;
                       #Step := 40;
                   END_IF;
                   ;
                   ;
                   ;
               END_IF;








               ;

              //Reject Logic 
           31:
               #Motor_Run := FALSE;
               #Pusher_Extend := TRUE;
               IF #Is_Pusher_Extended THEN
                   #Pusher_Extend := FALSE;
                   #Pusher_Release := TRUE;
                   #Step := 32;
               END_IF;
               ;

           32:
               #Motor_Run := FALSE;
               IF #Is_Pusher_Released THEN
                   #Pusher_Extend := FALSE;
                   #Pusher_Release := FALSE;
                   #Step := 33;
               END_IF;
               ;
               ;

           33:
               #Motor_Run := FALSE;

               //when Reject conveyor Sensor on and data transfer done than make it to step:=0
               IF #Reject_Conveyor_Step = 20 THEN
                   #Step := 0;
               END_IF;


               ;
           40:
               #Motor_Run := TRUE;

               IF NOT #Own_Sensor  THEN

                   #Motor_Run := FALSE;
                   #Step := 50;


               END_IF;






               ;
           50://reset to zero and ready for pick
               #Motor_Run := FALSE;
               IF #Is_Entry_Conveyor THEN
                   #Step := 0;

               ELSIF #Next_Conveyor_Step = 30 THEN //Verify Data transfer done,
                   #Motor_Run := FALSE;
                   #Step := 0;
               END_IF;
               ;
               ;



       END_CASE;

       ;
   ELSE
       #Motor_Run := FALSE;
       #Pusher_Extend := FALSE;
       #Pusher_Release := FALSE;
       #Jam_Detection_Timer(IN := FALSE,
                            PT := T#6s);

       IF #Reset & NOT #Own_Sensor & NOT #Auto THEN
           #Step := 0;
           #Jam_Enable := 0;
           #Jam_Detection_Timer(IN := FALSE,
                                PT := T#6s);
           ;
       END_IF;
   END_IF;
END_FUNCTION_BLOCK

FUNCTION_BLOCK "Arm_Pick_&_Place"   // FB2, SCL
{ S7_Optimized_Access := 'TRUE' }
VERSION : 0.1
   VAR_INPUT
      Ready_For_Pick : Bool;
      Going_Down : Bool;
      Going_Extend : Bool;
      Start : Bool;
      Reset : Bool;
      Rotating : Bool;
   END_VAR
   VAR_OUTPUT
      Go_Down : Bool;
      Grab : Bool;
      Go_Left : Bool;
      Go_Right : Bool;
      Go_Extend : Bool;
   END_VAR
   VAR RETAIN
      "Step" : Int;
   END_VAR
BEGIN

   IF #Start THEN


   CASE #Step OF
       0: //Going Down
           #Go_Right := FALSE;
           #Go_Left := FALSE;
           IF  #Ready_For_Pick & NOT #Rotating & NOT #Going_Extend  THEN
               #Go_Down := TRUE;
               #Step := 1;
           END_IF;
       1: //Grab
           #Go_Down := TRUE;
           IF NOT #Going_Down THEN
               #Go_Down := TRUE;
               #Grab := TRUE;
              #Step := 2;
           END_IF;
           ;
       2: //Going Up
           #Grab := TRUE;
           #Go_Down := FALSE;
           #Step := 3;
           ;

       3: //Moving Left && Extending Arm 
           #Grab := TRUE;
           IF NOT #Going_Down THEN
               #Go_Left := TRUE;
               #Go_Extend := TRUE;
               #Step := 4;
           END_IF;

           ;
       4:// Now Go down
           #Grab := TRUE;
           //#Go_Left := TRUE;
           #Go_Extend := TRUE;
           IF NOT #Rotating & NOT #Going_Extend THEN
               #Go_Down := TRUE;
               #Step := 5;
           END_IF;

           ;
       5:// Now left box
           #Go_Down := TRUE;
           IF NOT #Going_Down THEN
               #Go_Down := TRUE;
               #Grab := FALSE;
               #Step := 6;
           END_IF;

           ;
       6://Home position
           #Go_Down := FALSE;
           IF NOT #Going_Down THEN
               #Go_Extend := FALSE;
               #Go_Right := TRUE;
               #Step := 0;
           END_IF;

           ;

     (*  ELSE
           #Go_Extend := FALSE;
           #Go_Right := FALSE;
           #Go_Down := FALSE;
           #Go_Left := FALSE;
           #Grab := FALSE;
           ;
   *)
   END_CASE;

   ELSE
       #Go_Extend := FALSE;
       #Go_Right := FALSE;
       #Go_Down := FALSE;
       #Go_Left := FALSE;
       #Grab := FALSE;
       IF #Reset  THEN
           #Step := 0;
           ;
       END_IF;
   END_IF;
END_FUNCTION_BLOCK

FUNCTION_BLOCK "Reject_Conveyor_Control"   // FB3, SCL
{ S7_Optimized_Access := 'TRUE' }
VERSION : 0.1
   VAR_INPUT
      Decision_Conveyor_Step : Int;
      Start : Bool;
      Reset : Bool;
      Own_Sensor : Bool;
      Prev_Box_Data : "UDT_Box_Data";
   END_VAR
   VAR_OUTPUT
      Motor_Run : Bool;
   END_VAR
   VAR_IN_OUT
      Reject_Boxes : Int;
      Reject_Total_Weight : Real;
   END_VAR
   VAR
      "Step" : Int;
      My_Box_Data : "UDT_Box_Data";
   END_VAR
BEGIN
   IF #Start THEN
       CASE #Step OF
           0:  
               #Motor_Run := FALSE;
               IF #Decision_Conveyor_Step = 31 & NOT #Own_Sensor THEN
                   #Motor_Run := TRUE;
                   #Step := 10;
                   ;
               END_IF;
               ;
           10:
               #Motor_Run := TRUE;
               IF #Own_Sensor THEN
                   #Motor_Run := FALSE;
                   //Directly Update Reject Count +1, And save Weight +, Then no needed to transfer data..
                   "FC_BoxData_Transfer"(Prev_Box_Data := #Prev_Box_Data,
                                         My_Box_Data => #My_Box_Data);
               #Step:=20;
               END_IF;
               ;

           20:
               #Motor_Run := FALSE;
               IF #Own_Sensor THEN
                   #Motor_Run := TRUE;
                   #Step := 30;
               END_IF;
               ;
               ;
           30:
               #Motor_Run := TRUE;
               IF NOT #Own_Sensor THEN
                   #Motor_Run := FALSE;
                   #Reject_Boxes := #Reject_Boxes + 1;
                   #Reject_Total_Weight := (#Reject_Total_Weight + #My_Box_Data.Weight);
                   #Step := 0;
               END_IF;
               ;
               ;
       END_CASE;


   ELSE
       #Motor_Run := FALSE;
       IF #Reset & NOT #Own_Sensor THEN

           #Step := 0;
           ;
       END_IF;
   END_IF;
END_FUNCTION_BLOCK

// folder: 03_Library_FCs

FUNCTION "FC_BoxData_Transfer" : Void   // FC3, SCL
{ S7_Optimized_Access := 'TRUE' }
VERSION : 0.1
   VAR_INPUT
      Prev_Box_Data : "UDT_Box_Data";
   END_VAR
   VAR_OUTPUT
      My_Box_Data : "UDT_Box_Data";
   END_VAR
BEGIN
   #My_Box_Data.BoxId := #Prev_Box_Data.BoxId;
   #My_Box_Data.Weight := #Prev_Box_Data.Weight;
   #My_Box_Data.Status := #Prev_Box_Data.Status;
END_FUNCTION

FUNCTION "FC_WeighScale_Data_Transfer" : Void   // FC4, SCL
{ S7_Optimized_Access := 'TRUE' }
VERSION : 0.1
   VAR_INPUT
      Actual_Data : "UDT_Box_Real_Data";
   END_VAR
   VAR_OUTPUT
      My_Box_Data : "UDT_Box_Data";
   END_VAR
BEGIN
   #My_Box_Data.Weight := #Actual_Data.Actual_Weight_Value;
   #My_Box_Data.BoxId := #Actual_Data.Current_Box_ID + 1;

   IF #My_Box_Data.Weight >= #Actual_Data.Accept_Limit_Low & #My_Box_Data.Weight <=#Actual_Data.Accept_Limit_High THEN
       #My_Box_Data.Status := TRUE;
   ELSE
       #My_Box_Data.Status := FALSE;
      END_IF;
END_FUNCTION

FUNCTION "Jam_Detection" : Void   // FC5, SCL
{ S7_Optimized_Access := 'TRUE' }
VERSION : 0.1
   VAR_INPUT
      Start : Bool;
      "Ack ALL" : Bool;
      Entry_OL_Detected : Bool;
      Weigh_OL_Detected : Bool;
      Decision_OL_Detected : Bool;
      Reject_OL_Detected : Bool;
      Exit_OL_Detected : Bool;
   END_VAR
   VAR_OUTPUT
      Enable_Entry : Bool;
      Enable_Weigh : Bool;
      Enable_Decision : Bool;
      Enable_Reject : Bool;
      Enable_Exit : Bool;
      Enable_Robot : Bool;
      System_Running : Bool;
   END_VAR
   VAR_IN_OUT
      Motor_Overload : Struct
         OL_EntryMotor : "UDT_Alarm";
         OL_WeighMotor : "UDT_Alarm";
         OL_DecisionMotor : "UDT_Alarm";
         OL_RejectMotor : "UDT_Alarm";
         OL_ExitMotor : "UDT_Alarm";
      END_STRUCT;
      Jam_Alarm : Struct
         Jam_EntryMotor : "UDT_Alarm";
         Jam_WeighMotor : "UDT_Alarm";
         Jam_DecisionMotor : "UDT_Alarm";
         Jam_RejectMotor : "UDT_Alarm";
         Jam_ExitMotor : "UDT_Alarm";
      END_STRUCT;
      Pusher_Alarm : Struct
         Pusher_Stuck_Extended : "UDT_Alarm";
         Pusher_Stuck_Retracted : "UDT_Alarm";
      END_STRUCT;
      Jam_Detected : Struct
         Entry_Jam_Detected : Bool;
         Weigh_Jam_Detected : Bool;
         Decision_Jam_Detected : Bool;
         Reject_Jam_Detected : Bool;
         Exit_Jam_Detected : Bool;
      END_STRUCT;
   END_VAR
   VAR_TEMP
      Current_Time : DTL;
   END_VAR
BEGIN
   IF #"Ack ALL" THEN

       //Forced Cleared as it's Software generated...
       #Jam_Detected.Entry_Jam_Detected := FALSE;
       #Jam_Detected.Weigh_Jam_Detected := FALSE;
       #Jam_Detected.Decision_Jam_Detected := FALSE;
       #Jam_Detected.Reject_Jam_Detected := FALSE;
       #Jam_Detected.Exit_Jam_Detected := FALSE;

       //Reset Entry Conveyor
       IF #Jam_Alarm.Jam_EntryMotor.Cleared THEN
           #Jam_Alarm.Jam_EntryMotor.Active := FALSE;
           #Jam_Alarm.Jam_EntryMotor.Acknowledge := TRUE;

       END_IF;

       //Reset Weigh Conveyor
       IF #Jam_Alarm.Jam_WeighMotor.Cleared THEN
           #Jam_Alarm.Jam_WeighMotor.Active := FALSE;
           #Jam_Alarm.Jam_WeighMotor.Acknowledge := TRUE;
       END_IF;

       //Reset Decision Conveyor
       IF #Jam_Alarm.Jam_DecisionMotor.Cleared THEN
           #Jam_Alarm.Jam_DecisionMotor.Active := 0;
           #Jam_Alarm.Jam_DecisionMotor.Acknowledge := 1;
       END_IF;

       //Reset Reject Conveyor
       IF #Jam_Alarm.Jam_RejectMotor.Cleared THEN
           #Jam_Alarm.Jam_RejectMotor.Active := 0;
           #Jam_Alarm.Jam_RejectMotor.Acknowledge := 1;
       END_IF;

       //Reset Exit Conveyor
       IF #Jam_Alarm.Jam_ExitMotor.Cleared THEN
           #Jam_Alarm.Jam_ExitMotor.Active := 0;
           #Jam_Alarm.Jam_ExitMotor.Acknowledge := 1;
       END_IF;




   END_IF;





       #Enable_Robot := TRUE;
       #System_Running := TRUE;

       //Entry Logic
       #Enable_Entry := NOT #Jam_Detected.Entry_Jam_Detected & NOT #Entry_OL_Detected & NOT #Jam_Alarm.Jam_EntryMotor.Active & NOT #Jam_Alarm.Jam_WeighMotor.Active & NOT #Jam_Alarm.Jam_DecisionMotor.Active & NOT #Jam_Alarm.Jam_ExitMotor.Active;

       #Enable_Weigh := NOT #Jam_Detected.Weigh_Jam_Detected & NOT #Weigh_OL_Detected & NOT #Jam_Alarm.Jam_WeighMotor.Active & NOT #Jam_Alarm.Jam_DecisionMotor.Active & NOT #Jam_Alarm.Jam_ExitMotor.Active ;

       #Enable_Decision := NOT #Jam_Detected.Decision_Jam_Detected & NOT #Decision_OL_Detected & NOT #Jam_Alarm.Jam_DecisionMotor.Active & NOT #Jam_Alarm.Jam_ExitMotor.Active ;

       #Enable_Exit := NOT #Jam_Detected.Exit_Jam_Detected & NOT #Exit_OL_Detected & NOT #Jam_Alarm.Jam_ExitMotor.Active;

       #Enable_Reject := NOT #Jam_Detected.Reject_Jam_Detected & NOT #Reject_OL_Detected & NOT #Jam_Alarm.Jam_RejectMotor.Active;


       //Set Alarm Logic
       //Entry Jam
       IF #Jam_Detected.Entry_Jam_Detected THEN

           IF NOT #Jam_Alarm.Jam_EntryMotor.Active THEN

               #Enable_Entry := FALSE;
               #Jam_Alarm.Jam_EntryMotor.Active := TRUE;
               #Jam_Alarm.Jam_EntryMotor.TimeStamp := #Current_Time;
               #Jam_Alarm.Jam_EntryMotor.Cleared := FALSE;
           END_IF;

       ELSE
           IF #Jam_Alarm.Jam_EntryMotor.Active & NOT #Jam_Alarm.Jam_EntryMotor.Cleared THEN
               #Jam_Alarm.Jam_EntryMotor.Cleared := TRUE;




           END_IF;


       END_IF;



       //Weigh Jam
       IF #Jam_Detected.Weigh_Jam_Detected THEN

           IF NOT #Jam_Alarm.Jam_WeighMotor.Active THEN

               #Enable_Entry := FALSE;
               #Enable_Weigh := FALSE;
               #Jam_Alarm.Jam_WeighMotor.Active := TRUE;
               #Jam_Alarm.Jam_WeighMotor.TimeStamp := #Current_Time;
               #Jam_Alarm.Jam_WeighMotor.Cleared := 0;

           END_IF;

       ELSE

           IF #Jam_Alarm.Jam_WeighMotor.Active & NOT #Jam_Alarm.Jam_WeighMotor.Cleared THEN

               #Jam_Alarm.Jam_WeighMotor.Cleared := 1;





           END_IF;


       END_IF;








       //Decision Jam
       IF #Jam_Detected.Decision_Jam_Detected THEN


           IF NOT #Jam_Alarm.Jam_DecisionMotor.Active THEN



               #Enable_Entry := FALSE;
               #Enable_Weigh := FALSE;
               #Enable_Decision := FALSE;
               #Jam_Alarm.Jam_DecisionMotor.Active := TRUE;
               #Jam_Alarm.Jam_DecisionMotor.TimeStamp := #Current_Time;
               #Jam_Alarm.Jam_DecisionMotor.Cleared := 0;

           END_IF;

       ELSE

           IF #Jam_Alarm.Jam_DecisionMotor.Active & NOT #Jam_Alarm.Jam_DecisionMotor.Cleared THEN
               #Jam_Alarm.Jam_DecisionMotor.Cleared := 1;


           END_IF;



       END_IF;




       //Exit Jam
       IF #Jam_Detected.Exit_Jam_Detected THEN

           IF NOT #Jam_Alarm.Jam_ExitMotor.Active THEN

               #Enable_Entry := FALSE;
               #Enable_Weigh := FALSE;
               #Enable_Decision := FALSE;
               #Enable_Exit := FALSE;
               #Jam_Alarm.Jam_ExitMotor.Active := TRUE;
               #Jam_Alarm.Jam_ExitMotor.TimeStamp := #Current_Time;
               #Jam_Alarm.Jam_ExitMotor.Cleared := 0;

           END_IF;

       ELSE
           IF #Jam_Alarm.Jam_ExitMotor.Active & NOT #Jam_Alarm.Jam_ExitMotor.Cleared THEN
               #Jam_Alarm.Jam_ExitMotor.Cleared := 1;



           END_IF;


       END_IF;

       //Reject Jam
       IF #Jam_Detected.Reject_Jam_Detected THEN

           IF NOT #Jam_Alarm.Jam_RejectMotor.Active THEN


               #Enable_Reject := FALSE;
               #Jam_Alarm.Jam_RejectMotor.Active := TRUE;
               #Jam_Alarm.Jam_RejectMotor.TimeStamp := #Current_Time;
               #Jam_Alarm.Jam_RejectMotor.Cleared := 0;
           END_IF;

       ELSE
           IF #Jam_Alarm.Jam_RejectMotor.Active & NOT #Jam_Alarm.Jam_RejectMotor.Cleared THEN
               #Jam_Alarm.Jam_RejectMotor.Cleared := 1;
           END_IF;

       END_IF;
END_FUNCTION

FUNCTION "FC_HMI_Interface" : Void   // FC6, SCL
{ S7_Optimized_Access := 'TRUE' }
VERSION : 0.1
   VAR_INPUT
      OL_Entry : Bool;
      OL_Weigh : Bool;
      OL_Decision : Bool;
      OL_Exit : Bool;
      OL_Reject : Bool;
      Jam_Entry : Bool;
      Jam_Weigh : Bool;
      Jam_Decision : Bool;
      Jam_Exit : Bool;
      Jam_Reject : Bool;
      E_Stop : Bool;
      Batch_Boxes : Int;
      Accept_Boxes : Int;
   END_VAR
   VAR_OUTPUT
      Jam_Alarm : Word;
      OL_Alarm : Word;
      System_Alarm : Word;
   END_VAR
BEGIN


   // Clear all bits first
   #Jam_Alarm := WORD#0;

   // Then set bits
   #Jam_Alarm.%X0 := #Jam_Entry;
   #Jam_Alarm.%X1 := #Jam_Weigh;
   #Jam_Alarm.%X2 := #Jam_Decision;
   #Jam_Alarm.%X3 := #Jam_Exit;
   #Jam_Alarm.%X4 := #Jam_Reject;

   #System_Alarm := WORD#0;
   #System_Alarm.%X0 := NOT #E_Stop;
   #System_Alarm.%X1 := #Batch_Boxes <= #Accept_Boxes ;

   #OL_Alarm := WORD#0;

   #OL_Alarm.%X0 := #OL_Entry;
   #OL_Alarm.%X1 := #OL_Weigh;
   #OL_Alarm.%X2 := #OL_Decision;
   #OL_Alarm.%X3 := #OL_Exit;
   #OL_Alarm.%X4 := #OL_Reject;
END_FUNCTION

FUNCTION "FC_Startup" : Void   // FC7, SCL
{ S7_Optimized_Access := 'TRUE' }
VERSION : 0.1
   VAR_OUTPUT
      Accept_Boxes : Int;
      Reject_Boxes : Int;
      Accept_Total_Weight : Real;
      Reject_Total_Weight : Real;
      Batch_Boxes : Int;
      Low_Limit_Tag : Real;
      High_Limit_Tag : Real;
   END_VAR
   VAR_IN_OUT
      Jam_Detected : Struct
         Entry_Jam_Detected : Bool;
         Weigh_Jam_Detected : Bool;
         Decision_Jam_Detected : Bool;
         Reject_Jam_Detected : Bool;
         Exit_Jam_Detected : Bool;
      END_STRUCT;
   END_VAR
BEGIN
   #Accept_Boxes := 0;
   #Reject_Boxes := 0;
   #Accept_Total_Weight := 0.0;
   #Reject_Total_Weight := 0.0;
   #Batch_Boxes := 100;
   #Low_Limit_Tag := 3.0;
   #High_Limit_Tag := 6.0;


   #Jam_Detected.Entry_Jam_Detected := 0;
   #Jam_Detected.Weigh_Jam_Detected := 0;
   #Jam_Detected.Decision_Jam_Detected := 0;
   #Jam_Detected.Reject_Jam_Detected := 0;
   #Jam_Detected.Exit_Jam_Detected := 0;
END_FUNCTION

FUNCTION "FC_Clear_O/P" : Void   // FC8, SCL
{ S7_Optimized_Access := 'TRUE' }
VERSION : 0.1
   VAR_IN_OUT
      Output : Struct
         Q_Motor_Entry : Bool;
         Q_Motor_Weigh : Bool;
         Q_Motor_Decision : Bool;
         Q_Motor_reject : Bool;
         Q_Motor_Exit : Bool;
         Q_Pusher_Extend : Bool;
         Q_Pusher_Release : Bool;
         Q_Signal_Red : Bool;
         Q_Signal_Yellow : Bool;
         Q_Signal_Green : Bool;
         Q_Buzzer : Bool;
         Q_Robot_Extend_X : Bool;
         Q_Robot_Down_Z : Bool;
         Q_Robot_Grab : Bool;
         Q_Robot_Rotate_CW : Bool;
         Q_Robot_Rotate_CCW : Bool;
      END_STRUCT;
   END_VAR
BEGIN
   #Output.Q_Motor_Entry := 0;
   #Output.Q_Motor_Weigh := 0;
   #Output.Q_Motor_Decision := 0;
   #Output.Q_Motor_reject := 0;
   #Output.Q_Motor_Exit := 0;
   #Output.Q_Pusher_Extend := 0;
   #Output.Q_Pusher_Release := 0;
   #Output.Q_Robot_Extend_X := 0;
   #Output.Q_Robot_Down_Z := 0;
   #Output.Q_Robot_Grab := 0;
   #Output.Q_Robot_Rotate_CW := 0;
   #Output.Q_Robot_Rotate_CCW := 0;
END_FUNCTION

FUNCTION "FC_Signal_Lamp" : Void   // FC9, FBD
{ S7_Optimized_Access := 'TRUE' }
VERSION : 0.1
   VAR_INPUT
      I_PB_Emergency : Bool;
      M_START : Bool;
      Clock : Bool;
   END_VAR
   VAR_OUTPUT
      Q_Signal_Red : Bool;
      Q_Signal_Green : Bool;
   END_VAR
   VAR_IN_OUT
      Jam_Alarm : Struct
         Jam_EntryMotor : "UDT_Alarm";
         Jam_WeighMotor : "UDT_Alarm";
         Jam_DecisionMotor : "UDT_Alarm";
         Jam_RejectMotor : "UDT_Alarm";
         Jam_ExitMotor : "UDT_Alarm";
      END_STRUCT;
   END_VAR
   VAR_TEMP
      Red_Light : Bool;
   END_VAR
BEGIN

REGION Network 1
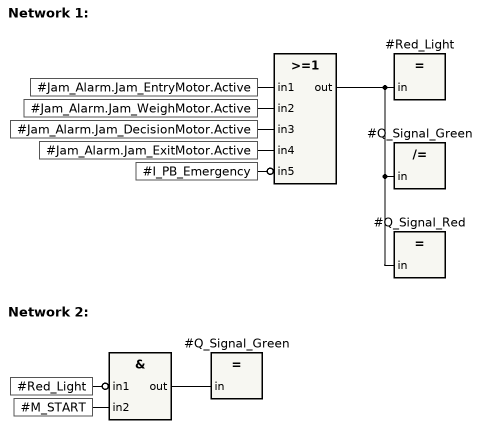
   #Red_Light := #Jam_Alarm.Jam_EntryMotor.Active OR #Jam_Alarm.Jam_WeighMotor.Active OR #Jam_Alarm.Jam_DecisionMotor.Active OR #Jam_Alarm.Jam_ExitMotor.Active OR NOT #I_PB_Emergency;
   #Q_Signal_Green := NOT #Red_Light;
   #Q_Signal_Red := #Red_Light;
END_REGION

REGION Network 2
   #Q_Signal_Green := NOT #Red_Light AND #M_START;
END_REGION
END_FUNCTION

FUNCTION "MHJ-PLC-Lab-Function-S71200" : Void   // FC9000, SCL
{ S7_Optimized_Access := 'TRUE' }
VERSION : 0.1
   VAR_TEMP
      rdTimeReturn : Int;
      outputTime : DTL;
      SyncVal : Byte;
      forVal : Int;
      forVal_2 : Int;
      Value : Byte;
   END_VAR
   VAR CONSTANT
      CompVal : Byte := 16#34;
      Value_01 : Byte := 16#11;
      Value_01_DW : DWord := 16#A165_D992;
      Value_02_DW : DWord := 16#58BE_4401;
   END_VAR
BEGIN

   #Value:=PEEK(area := 16#82,
        dbNumber := 0,
        byteOffset := 511);
   #Value := #Value + 1;

   POKE(area := 16#82,
        dbNumber := 0,
        byteOffset := 511,
        value := #Value);

   POKE(area:=16#81,
        dbNumber:=0,
        byteOffset:=1016,
        value:=#Value_01_DW);
   POKE(area := 16#81,
        dbNumber := 0,
        byteOffset := 1020,
        value := #Value_02_DW);

   POKE(area := 16#81,
        dbNumber := 0,
        byteOffset := 511,
        value := B#16#00);

   FOR #forVal := 0 TO 500 DO
       FOR #forVal_2:=0 TO 10 DO
           #rdTimeReturn:=RD_SYS_T(#outputTime);
           #rdTimeReturn := WR_SYS_T(#outputTime);
           #rdTimeReturn := RD_SYS_T(#outputTime);
           #rdTimeReturn := WR_SYS_T(#outputTime);
       END_FOR;
       #SyncVal:= PEEK(area := 16#81,
                      dbNumber := 0,
                      byteOffset := 511);
       IF #SyncVal = #CompVal THEN
          GOTO M_1;
       END_IF;
   END_FOR;
   RETURN;

   M_1:
   POKE(area := 16#81,
        dbNumber := 0,
        byteOffset := 511,
        value := B#16#0);
END_FUNCTION

// folder: 06_IO_Mapping

FUNCTION "FC_Input_Mapping" : Void   // FC1, SCL
{ S7_Optimized_Access := 'TRUE' }
VERSION : 0.1
BEGIN

   "DB_IO_Mapping".Input.I_PB_Start := "I_PB_Start";
   "DB_IO_Mapping".Input.I_PB_Stop := "I_PB_Stop";
   "DB_IO_Mapping".Input.I_PB_Emergency := "I_PB_Emergency";
   "DB_IO_Mapping".Input.I_PB_Reset := "I_PB_Reset";
   "DB_IO_Mapping".Input.I_PB_Auto := "I_PB_Auto";
   "DB_IO_Mapping".Input.I_Sensor_Entry := "I_Sensor_Entry";
   "DB_IO_Mapping".Input.I_Sensor_Weigh := "I_Sensor_Weigh";
   "DB_IO_Mapping".Input.I_Sensor_Decision := "I_Sensor_Decision";
   "DB_IO_Mapping".Input.I_Sensor_Reject := "I_Sensor_Reject";
   "DB_IO_Mapping".Input.I_Sensor_Exit := "I_Sensor_Exit";
   "DB_IO_Mapping".Input.I_Pusher_Extend := "I_Pusher_Extend";
   "DB_IO_Mapping".Input.I_Pusher_Released := "I_Pusher_Released";
   "DB_IO_Mapping".Input.I_OL_EntryMotor := "I_OL_EntryMotor";
   "DB_IO_Mapping".Input.I_OL_WeighMotor := "I_OL_WeighMotor";
   "DB_IO_Mapping".Input.I_OL_DecideMotor := "I_OL_DecideMotor";
   "DB_IO_Mapping".Input.I_OL_RejectMotor := "I_OL_RejectMotor";
   "DB_IO_Mapping".Input.I_OL_ExitMotor := "I_OL_ExitMotor";
   "DB_IO_Mapping".Input.I_Robot_Detect := "I_Robot_Detect";
   "DB_IO_Mapping".Input.I_Robot_Moving_X := "I_Robot_Moving_X";
   "DB_IO_Mapping".Input.I_Robot_Moving_Z := "I_Robot_Moving_Z";
   "DB_IO_Mapping".Input.I_Robot_Rotating := "I_Robot_Rotating";

   "DB_IO_Mapping".Input.IW_Weight_Loadcell := "IW_Weight_Loadcell";
   IF "DB_IO_Mapping".Input.IW_Weight_Loadcell > 6.0 THEN
       "DB_Batch_Data".Real_Box_Data.Actual_Weight_Value := 7.5;
   ELSE
       "DB_Batch_Data".Real_Box_Data.Actual_Weight_Value := 4.0;
   END_IF;



   "DB_Batch_Data".Real_Box_Data.Accept_Limit_Low := "DB_Batch_Data".Low_Limit_Tag;
   "DB_Batch_Data".Real_Box_Data.Accept_Limit_High := "DB_Batch_Data".High_Limit_Tag;

   "DB_Batch_Data".Low_Limit_Tag_1 := "DB_Batch_Data".Low_Limit_Tag;
   "DB_Batch_Data".High_Limit_Tag_1 := "DB_Batch_Data".High_Limit_Tag;

   (*
   "DB_IO_Mapping".Input.I_PB_Start := "I_PB_Start";
   "DB_IO_Mapping".Input.I_PB_Stop := "I_PB_Stop";
   "DB_IO_Mapping".Input.I_PB_Emergency := "I_PB_Emergency";
   "DB_IO_Mapping".Input.I_PB_Reset := "I_PB_Reset";
   "DB_IO_Mapping".Input.I_PB_Auto := "I_PB_Auto";
   "DB_IO_Mapping".Input.I_Sensor_Entry := "I_Sensor_Entry";
   "DB_IO_Mapping".Input.I_Sensor_Weigh := "I_Sensor_Weigh";
   "DB_IO_Mapping".Input.I_Sensor_Decision := "I_Sensor_Decision";
   "DB_IO_Mapping".Input.I_Sensor_Reject := "I_Sensor_Reject";
   "DB_IO_Mapping".Input.I_Sensor_Exit := "I_Sensor_Exit";
   "DB_IO_Mapping".Input.I_Pusher_Extend := "I_Pusher_Extend";
   "DB_IO_Mapping".Input.I_Pusher_Released := "I_Pusher_Released";
   *)
   //-------------------------------------------------------------
END_FUNCTION

FUNCTION "FC_Output_Mapping" : Void   // FC2, SCL
{ S7_Optimized_Access := 'TRUE' }
VERSION : 0.1
BEGIN

   "Q_Motor_Entry" := "DB_IO_Mapping".Output.Q_Motor_Entry;
   "Q_Motor_Weigh" := "DB_IO_Mapping".Output.Q_Motor_Weigh;
   "Q_Motor_Decision" := "DB_IO_Mapping".Output.Q_Motor_Decision;
   "Q_Motor_reject" := "DB_IO_Mapping".Output.Q_Motor_reject;
   "Q_Motor_Exit" := "DB_IO_Mapping".Output.Q_Motor_Exit;
   "Q_Pusher_Extend" := "DB_IO_Mapping".Output.Q_Pusher_Extend;
   "Q_Pusher_Release" := "DB_IO_Mapping".Output.Q_Pusher_Release;
   "Q_Signal_Red" := "DB_IO_Mapping".Output.Q_Signal_Red;
   "Q_Signal_Yellow" := "DB_IO_Mapping".Output.Q_Signal_Yellow;
   "Q_Signal_Green" := "DB_IO_Mapping".Output.Q_Signal_Green;
   "Q_Buzzer" := "DB_IO_Mapping".Output.Q_Buzzer;
   "Q_Robot_Extend_X" := "DB_IO_Mapping".Output.Q_Robot_Extend_X;
   "Q_Robot_Down_Z" := "DB_IO_Mapping".Output.Q_Robot_Down_Z;
   "Q_Robot_Grab" := "DB_IO_Mapping".Output.Q_Robot_Grab;
   "Q_Robot_Rotate_CW" := "DB_IO_Mapping".Output.Q_Robot_Rotate_CW;
   "Q_Robot_Rotate_CCW" := "DB_IO_Mapping".Output.Q_Robot_Rotate_CCW;
END_FUNCTION

(* ===== HMI "HMI_RT_1" =====
system functions are stored by id; their names below are inferred from use
connection "HMI_Connection_1": ETHERNET, SMART_S7_1200_OMS

HMI tags "Default tag table"
   "Small Box Selected" : Bool, internal
   "DB_Batch_Data_Batch_Boxes" : Int = PLC DB_Batch_Data.Batch_Boxes, 1 s
   "DB_Batch_Data_Accept_Total_Weight" : Real = PLC DB_Batch_Data.Accept_Total_Weight, 1 s
   "DB_Batch_Data_Low_Limit_Tag" : Real = PLC DB_Batch_Data.Low_Limit_Tag, 1 s
   "DB_Batch_Data_High_Limit_Tag" : Real = PLC DB_Batch_Data.High_Limit_Tag, 1 s
   "DB_Batch_Data_Accept_Boxes" : Int = PLC DB_Batch_Data.Accept_Boxes, 1 s
   "DB_Batch_Data_Reject_Boxes" : Int = PLC DB_Batch_Data.Reject_Boxes, 1 s
   "DB_Batch_Data_Reject_Total_Weight" : Real = PLC DB_Batch_Data.Reject_Total_Weight, 1 s
   "DB_Alarms_HMI_Alarm_Jam_Alarm" : Word = PLC DB_Alarms.HMI_Alarm.Jam_Alarm, 1 s
   "DB_Alarms_HMI_Alarm_OL_Alarm" : Word = PLC DB_Alarms.HMI_Alarm.OL_Alarm, 1 s
   "DB_Alarms_HMI_Alarm_System_Alarm" : Word = PLC DB_Alarms.HMI_Alarm.System_Alarm, 1 s
   "DB_Alarms_HMI_Ack_All" : Bool = PLC DB_Alarms.HMI_Ack_All, 1 s
   "Large Box Selected" : Bool, internal
   "DB_Batch_Data_Low_Limit_Tag_1" : Real = PLC DB_Batch_Data.Low_Limit_Tag_1, 1 s
   "DB_Batch_Data_High_Limit_Tag_1" : Real = PLC DB_Batch_Data.High_Limit_Tag_1, 1 s

discrete alarms
   1: 'Entry Conveyor Jam', class Errors, trigger "DB_Alarms_HMI_Alarm_Jam_Alarm" bit 0
   2: 'Weigh Conveyor Jam', class Errors, trigger "DB_Alarms_HMI_Alarm_Jam_Alarm" bit 1
   3: 'Decision Conveyor Jam', class Errors, trigger "DB_Alarms_HMI_Alarm_Jam_Alarm" bit 2
   4: 'Exit Conveyor Jam', class Errors, trigger "DB_Alarms_HMI_Alarm_Jam_Alarm" bit 3
   5: 'Reject Conveyor Jam', class Errors, trigger "DB_Alarms_HMI_Alarm_Jam_Alarm" bit 4
   6: 'Entry Conveyor Motor MPCB Tripped', class Errors, trigger "DB_Alarms_HMI_Alarm_OL_Alarm" bit 0
   7: 'Weigh Conveyor Motor MPCB Tripped', class Errors, trigger "DB_Alarms_HMI_Alarm_OL_Alarm" bit 1
   8: 'Decision Conveyor Motor MPCB Tripped', class Errors, trigger "DB_Alarms_HMI_Alarm_OL_Alarm" bit 2
   9: 'Exit Conveyor Motor MPCB Tripped', class Errors, trigger "DB_Alarms_HMI_Alarm_OL_Alarm" bit 3
   10: 'Reject Conveyor Motor MPCB Tripped', class Errors, trigger "DB_Alarms_HMI_Alarm_OL_Alarm" bit 4
   11: 'Emergency Switch Stop', class Errors, trigger "DB_Alarms_HMI_Alarm_System_Alarm" bit 0
   12: 'Batch Completed', class Warnings, trigger "DB_Alarms_HMI_Alarm_System_Alarm" bit 1
   13: 'CPU Time Error', class Errors, trigger "DB_Alarms_HMI_Alarm_System_Alarm" bit 2

recipe "Recipe_1": Lower Limit <- "DB_Batch_Data_Low_Limit_Tag", Higher Limit <- "DB_Batch_Data_High_Limit_Tag"

Template "Template_1" 800x480
   DateTimeField "HmiScreenItemData" at 695,25 size 105x25
   DateTimeField "HmiScreenItemData_1" at 695,0 size 105x25
   GraphicView "Logo" at 0,0 size 91x51; Picture "Logo of HMI_1"

screen "Root screen" 800x480, template "Template_1"
   on GenerateScreen: SetTag("Small Box Selected", 1)
   IOField "I/O field_1" at 257,114 size 96x38; FormatPattern s999
      ProcessValue <- "DB_Batch_Data_Batch_Boxes"
   TextField "Text field_1" at 84,118 size 166x32; Text 'Set Batch Box'
   IOField "I/O field_4" at 629,154 size 100x50; FormatPattern s99999
      ProcessValue <- "DB_Batch_Data_Reject_Boxes"
   IOField "I/O field_5" at 457,154 size 100x50; FormatPattern s99999
      ProcessValue <- "DB_Batch_Data_Accept_Boxes"
   TextField "Text field_4" at 626,111 size 97x25; Text 'Reject Box'
   TextField "Text field_5" at 456,111 size 101x25; Text 'Accept Box'
   IOField "I/O field_6" at 629,254 size 100x50; FormatPattern s999999999.999
      ProcessValue <- "DB_Batch_Data_Reject_Total_Weight"
   IOField "I/O field_7" at 457,254 size 100x50; FormatPattern s999999999.999
      ProcessValue <- "DB_Batch_Data_Accept_Total_Weight"
   TextField "Text field_6" at 617,221 size 125x25; Text 'Reject Weight'
   TextField "Text field_7" at 440,221 size 129x25; Text 'Accept Weight'
   TextField "Text field_8" at 117,143 size 16x23; Text 'Text'
   Button "Button_1" at 86,166 size 166x32; TextOff 'Select Small Box'
      on Press: SetBit("Small Box Selected"); ResetBit("Large Box Selected"); function_eba64363(1, U 1, 1, N)
   Button "Button_2" at 84,212 size 168x32; TextOff 'Select Large Box'
      on Press: SetBit("Large Box Selected"); ResetBit("Small Box Selected"); function_eba64363(1, U 2, 1, N)
   Button "Button_3" at 668,415 size 100x45; TextOff 'Alarm'
      on Press: ActivateScreen("Alarm_Screen", 0)
   Circle "Circle_1" at 289,169 size 25x25
      Appearance <- "Small Box Selected"
   Circle "Circle_2" at 289,215 size 25x25
      Appearance <- "Large Box Selected"
   TextField "Text field_2" at 78,289 size 214x28; Text 'Acceptable Weight Range'
   IOField "I/O field_2" at 66,313 size 97x49; FormatPattern s999999999.999
      ProcessValue <- "DB_Batch_Data_Low_Limit_Tag_1"
   TextField "Text field_3" at 164,325 size 26x23; Text 'To'
   IOField "I/O field_3" at 189,313 size 99x49; FormatPattern s999999999.999
      ProcessValue <- "DB_Batch_Data_High_Limit_Tag_1"
   TextField "Text field_9" at 106,0 size 563x68; Text 'Home Screen'

screen "Alarm_Screen" 800x480, template "Template_1"
   AlarmView "Alarm view_1" at 31,69 size 736x337
   Button "Button_1" at 665,427 size 100x45; TextOff 'Ack All'
      on Press: SetBit("DB_Alarms_HMI_Ack_All")
      on Release: ResetBit("DB_Alarms_HMI_Ack_All")
   Button "Button_4" at 34,427 size 100x45; TextOff 'Home'
      on Press: ActivateScreen("Root screen", 0)
   TextField "Text field_9" at 104,0 size 600x68; Text 'Alarm Screen'
*)